INTERFACE I_BurnerControlEcoFlamV2 EXTENDS I_BurnerControlEcoFlam

METHOD MR_Reset : BOOL
VAR_INPUT
END_VAR
END_METHOD

PROPERTY Ref_poReset : REFERENCE TO fb_digitalOutput
GET
END_GET
END_PROPERTY

END_INTERFACE

(* stored: Version 1.1.0.1, ProductVersion 3.1.4024.12
   Itf I_BurnerControlEcoFlamV2: Id {07149acc-c85c-464c-8f57-bfbf2ddbcf90}
   Method MR_Reset: Id {8d5a4947-370d-4c23-bbd6-607c986532eb}
   Property Ref_poReset: Id {567f1aac-6c26-4788-8478-e64c8db0593e}
   Get Get: Id {a06ad692-2b46-424f-8354-a79b78fa33a2} *)
